FUNCTION_BLOCK ParameterSet
VAR_INPUT
END_VAR
VAR_OUTPUT
END_VAR
VAR
	m_idx: UINT := ResiConst.ARR_MIN;
	m_parameters : ARRAY [ResiConst.ARR_MIN..ResiConst.PARAMS_ARR_MAX] OF SNamedValue;
END_VAR

PROPERTY Parameters : ARRAY [ResiConst.ARR_MIN..ResiConst.PARAMS_ARR_MAX] OF SNamedValue
GET
Parameters := m_parameters;
END_GET
END_PROPERTY

METHOD Retrieve : SNamedValue
VAR_INPUT
	i_name: STRING;
END_VAR
VAR
	i: UINT;
	m_emptyParam: SNamedValue;
END_VAR
FOR i := ResiConst.ARR_MIN TO m_idx + 1 DO
	IF m_parameters[i].Name = i_name THEN
		Retrieve := m_parameters[i];
		RETURN;
	END_IF
END_FOR

Retrieve := m_emptyParam;
END_METHOD

METHOD SetParam_Binary : BOOL
VAR_INPUT
	i_key: STRING;
	i_value: BOOL;
END_VAR
VAR
	i: UINT;
	m_paramFound: BOOL;
END_VAR
FOR i := 0 TO m_idx BY 1 DO
	IF m_parameters[i].Name = i_key THEN
		m_parameters[i].DataType := EDataType.binary;
		m_parameters[i].Value.Binary := i_value;
		m_paramFound := TRUE;
	END_IF
END_FOR

IF NOT m_paramFound THEN
	m_idx := m_idx + 1;
	m_parameters[m_idx].DataType := EDataType.binary;
	m_parameters[m_idx].Value.Binary := i_value;
	m_parameters[m_idx].Name := i_key;
END_IF
END_METHOD

METHOD SetParam_Defined : BOOL
VAR_INPUT
	i_key: STRING;
	i_defined: BOOL;
END_VAR
VAR
	i: UINT;
	m_paramsFound: BOOL;	
END_VAR
FOR i := 0 TO m_idx BY 1 DO
	IF m_parameters[m_idx].Name = i_key THEN
		m_parameters[m_idx].Defined := i_defined;
		m_paramsFound := TRUE;
		SetParam_Defined := TRUE;
	END_IF
END_FOR

IF NOT m_paramsFound THEN
	SetParam_Defined := FALSE;
END_IF
END_METHOD

METHOD SetParam_Numeric : BOOL
VAR_INPUT
	i_key: STRING;
	i_value: LREAL;
END_VAR
VAR
	i: UINT;
	m_key: STRING;
	m_paramFound: BOOL;
END_VAR
FOR i := 0 TO m_idx BY 1 DO
	m_key := m_parameters[i].Name;
	IF m_key = i_key THEN
		m_parameters[i].DataType := EDataType.numeric;
		m_parameters[i].Value.Numeric := i_value;
		m_paramFound := TRUE;
	END_IF
END_FOR

IF NOT m_paramFound THEN
	m_idx := m_idx + 1;
	m_parameters[m_idx].DataType := EDataType.numeric;
	m_parameters[m_idx].Value.Numeric := i_value;
	m_parameters[m_idx].Name := i_key;
END_IF
END_METHOD

METHOD SetParam_String : BOOL
VAR_INPUT
	i_key: STRING;
	i_value: STRING;
END_VAR
VAR
	i: UINT;
	m_paramFound: BOOL;
END_VAR
FOR i := 0 TO m_idx BY 1 DO
	IF m_parameters[i].Name = i_key THEN
		m_parameters[i].DataType := EDataType.string_t;
		m_parameters[i].Value.String_t := i_value;
		m_paramFound := TRUE;
	END_IF
END_FOR

IF NOT m_paramFound THEN
	m_idx := m_idx + 1;
	m_parameters[m_idx].DataType := EDataType.string_t;
	m_parameters[m_idx].Value.String_t := i_value;
	m_parameters[m_idx].Name := i_key;
END_IF
END_METHOD

END_FUNCTION_BLOCK

(* stored: Version 1.1.0.1, ProductVersion 3.1.4024.9
   POU ParameterSet: Id {eb331099-ae97-4f32-aa88-df5977516e9d}, SpecialFunc None
   Property Parameters: Id {d1f2b1be-85ac-48db-ad72-e6b7ae4b9e3a}
   Get Get: Id {80978e2a-eb98-44f5-92a4-995ebdc61823}
   Method Retrieve: Id {5be741c3-bbce-45ed-a7fb-f3cef9e4ab38}
   Method SetParam_Binary: Id {72712b4e-6142-4af3-b5bd-214df5a17002}
   Method SetParam_Defined: Id {db6ebabb-bcc5-448f-bb5f-334b6d605963}
   Method SetParam_Numeric: Id {c64b80ec-0f11-4462-a080-1364db3674c8}
   Method SetParam_String: Id {49d2cf7c-4418-4dd7-ad0a-e586ed586998} *)
